FUNCTION_BLOCK SAMPLE_UINT (* Sample a single UINT *)
  (* Standard: 61499-1; Classification: Math; Function: Sampling; Type: UINT *)
  (* Version 0.1, 2008-06-25, JHC, Holobloc Inc, Updated to new implementation. *)
  (* Version 0.0, 2006-05-28, JHC, Holobloc Inc *)
  (* Compiler header: package fb.rt.math; *)
  (* Compiler classdef: public class SAMPLE_UINT extends ChangeSensor *)
  (* Compiler Java Sun JDK 1.5.0 *)
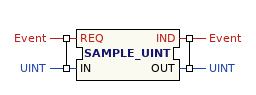
  EVENT_INPUT
    REQ WITH IN; (* Request to Sample *)
  END_EVENT
  EVENT_OUTPUT
    IND WITH OUT; (* Initial Sample or OUT changed *)
  END_EVENT
  VAR_INPUT
    IN : UINT; (* Data to Sample *)
  END_VAR
  VAR_OUTPUT
    OUT : UINT; (* Sampled Data *)
  END_VAR
END_FUNCTION_BLOCK
